PROGRAM MAIN
VAR
bChangeSeparatorToComma	: BOOL := TRUE;
P_TextModeWrite_WriteTrigger:BOOL:=FALSE;
P_TextModeWrite_WriteFilePath:T_MaxString := 'C:\Users\Administrator\Desktop\Pos.csv';
P_TextModeRead_ReadTrigger:BOOL:=FALSE;
P_TextModeRead_ReadFilePath:T_MaxString := 'C:\Users\Administrator\Desktop\Pos.csv';

CurrentJob: INT:= 0;//Job Code
CurrentJobState:STRING(80);//Say in which state

LAMP:BOOL;
POWER:BOOL;
Move_AB:BOOL;

SetPointGenEnable:ARRAY [0..5] OF MC_ExtSetPointGenEnable;
SetpointGenDisable:ARRAY [0..5] OF MC_ExtSetpointGenDisable;
SetPointGenEnable_output: ARRAY [0..5] OF ST_McOutputs;
SetPointGenDisable_output: ARRAY [0..5] OF ST_McOutputs;
enable:ARRAY [0..5] OF BOOL;
disable:ARRAY [0..5] OF BOOL;

position:ARRAY [0..5] OF LREAL;
velocity:ARRAY [0..5] OF LREAL;
direction:ARRAY [0..5] OF DINT;
acceleration:ARRAY [0..5] OF LREAL;

Pos_arr1:ARRAY[0..4999,0..5] OF LREAL;
i:INT;
FiFo_GetDimension: FiFoGetDimension;
fifo_display: STRING(255);

FiFo_GroupIntegrate1,FiFo_GroupIntegrate2,FiFo_GroupIntegrate3,FiFo_GroupIntegrate4,FiFo_GroupIntegrate6,FiFo_GroupIntegrate5: FiFoGroupIntegrate;
FiFo_SetChannelOverride:FiFoSetChannelOverride;
FiFo_Groupout1,FiFo_Groupout2,FiFo_Groupout3,FiFo_Groupout4,FiFo_Groupout5,FiFo_Groupout6,FiFo_Disintegrate,FiFo_Override_output:st_mcoutputs;
integrate_do:BOOL;
FiFo_GroupDisintegrate:FiFoGroupDisintegrate;

FiFo_Start:FiFoStart;
start_do:BOOL;
FiFo_Stop:FiFoStop;
stop_do:BOOL;
fifo_startoutput,fifo_stopoutput:st_mcoutputs;

FiFo_Write:FiFoWrite;
FIFO_write_do:BOOL;
FiFo_overWrite:FiFoOverwrite;
FIFO_overwrite_do:BOOL;
FIFO_write_output:st_mcoutputs;

END_VAR
VAR CONSTANT
	GlobalSetSpeed : ARRAY[0..5]OF LREAL:=[3200,3200,3200,3200,3200,3200];
END_VAR

IF bChangeSeparatorToComma THEN
	DEFAULT_CSV_FIELD_SEP := 16#2C;(* Comma ASCII code *)
ELSE
	DEFAULT_CSV_FIELD_SEP := 16#3B;(* Semicolon ASCII code *)
END_IF

IF FiFo_GetDimension.iNoOfAxes=6 AND FiFo_GetDimension.iNoOfFifoEntries=200 THEN
	fifo_display:='Parameters OK';
ELSE
	fifo_display:='Parameters Bad';
END_IF

//fifo();

GVL.LineMoveSpeed:=STRING_TO_LREAL(GVL.LineMoveSpeedString);
GVL.CMoveSpeed:=STRING_TO_LREAL(GVL.CMoveSpeedString);
GVL.OutMovePos[0]:=STRING_TO_LREAL(GVL.OutMovePosString[0]);
GVL.OutMovePos[1]:=STRING_TO_LREAL(GVL.OutMovePosString[1]);
GVL.OutMovePos[2]:=STRING_TO_LREAL(GVL.OutMovePosString[2]);
GVL.OutCMovePos[0]:=STRING_TO_LREAL(GVL.OutCMovePosString[0]);
GVL.OutCMovePos[1]:=STRING_TO_LREAL(GVL.OutCMovePosString[1]);
GVL.OutCMovePos[2]:=STRING_TO_LREAL(GVL.OutCMovePosString[2]);
GVL.MoveA[0]:=STRING_TO_LREAL(GVL.MoveAString[0])*24.995;
GVL.MoveA[1]:=STRING_TO_LREAL(GVL.MoveAString[1])*32.28;
GVL.MoveA[2]:=STRING_TO_LREAL(GVL.MoveAString[2])*49.845;
GVL.MoveA[3]:=STRING_TO_LREAL(GVL.MoveAString[3])*50.905;
GVL.MoveA[4]:=STRING_TO_LREAL(GVL.MoveAString[4])*80.34;
GVL.MoveA[5]:=STRING_TO_LREAL(GVL.MoveAString[5])*60.5;
GVL.OutActPos[0]:=-GVL.Axis[0].NcToPlc.ActPos/24.995;
GVL.OutActPos[1]:=-GVL.Axis[1].NcToPlc.ActPos/32.28;
GVL.OutActPos[2]:=GVL.Axis[2].NcToPlc.ActPos/49.845;
GVL.OutActPos[3]:=GVL.Axis[3].NcToPlc.ActPos/50.905;
GVL.OutActPos[4]:=GVL.Axis[4].NcToPlc.ActPos/80.34;
GVL.OutActPos[5]:=GVL.Axis[5].NcToPlc.ActPos/60.5;

IF GVL.ExtPosReady = FALSE THEN	
MC_ExtSetPointGenFeed(Position:=-GVL.OutActPos[0]*24.995,Velocity:= 0,Acceleration:=0,Direction:=1,Axis:=Axis[0]);	
MC_ExtSetPointGenFeed(Position:=-GVL.OutActPos[1]*32.28,Velocity:= 0,Acceleration:=0,Direction:=1,Axis:=Axis[1]);		
MC_ExtSetPointGenFeed(Position:=GVL.OutActPos[2]*49.845,Velocity:= 0,Acceleration:=0,Direction:=1,Axis:=Axis[2]);		
MC_ExtSetPointGenFeed(Position:=GVL.OutActPos[3]*50.905,Velocity:= 0,Acceleration:=0,Direction:=1,Axis:=Axis[3]);		
MC_ExtSetPointGenFeed(Position:=GVL.OutActPos[4]*80.34,Velocity:= 0,Acceleration:=0,Direction:=1,Axis:=Axis[4]);		
MC_ExtSetPointGenFeed(Position:=GVL.OutActPos[5]*60.5,Velocity:= 0,Acceleration:=0,Direction:=1,Axis:=Axis[5]);		
END_IF

CASE CurrentJob OF	
	0://None state
		AxisStopTrigger[0]:=FALSE;AxisStopTrigger[1]:=FALSE;AxisStopTrigger[2]:=FALSE;
		AxisStopTrigger[3]:=FALSE;AxisStopTrigger[4]:=FALSE;AxisStopTrigger[5]:=FALSE;
		AxisStop();//失能功能块
		
		JogFw[0]:=FALSE;JogFw[1]:=FALSE;JogFw[2]:=FALSE;JogFw[3]:=FALSE;JogFw[4]:=FALSE;JogFw[5]:=FALSE;
		JogBw[0]:=FALSE;JogBw[1]:=FALSE;JogBw[2]:=FALSE;JogBw[3]:=FALSE;JogBw[4]:=FALSE;JogBw[5]:=FALSE;
		Move_JOG();//失能功能块
		
		AxisMoveTrigger[0]:=FALSE;AxisMoveTrigger[1]:=FALSE;AxisMoveTrigger[2]:=FALSE;
		AxisMoveTrigger[3]:=FALSE;AxisMoveTrigger[4]:=FALSE;AxisMoveTrigger[5]:=FALSE;
		AxisMoveAbsoulte();//失能功能块
		
		Home[0]:=FALSE;Home[1]:=FALSE;Home[2]:=FALSE;
		Home[3]:=FALSE;Home[4]:=FALSE;Home[5]:=FALSE;
		Homing();//失能功能块	

		AxisResetTrigger[0]:=FALSE;AxisResetTrigger[1]:=FALSE;AxisResetTrigger[2]:=FALSE;
		AxisResetTrigger[3]:=FALSE;AxisResetTrigger[4]:=FALSE;AxisResetTrigger[5]:=FALSE;
		AxisReset();//失能功能块
		
		P_TextModeWrite_WriteTrigger:=FALSE;
		P_TextModeWrite();	
		P_TextModeRead_ReadTrigger:=FALSE;
		P_TextModeRead();//失能功能块
		
		SetPointGenEnable[0].Execute:=FALSE;SetPointGenEnable[1].Execute:=FALSE;
		SetPointGenEnable[2].Execute:=FALSE;SetPointGenEnable[3].Execute:=FALSE;
		SetPointGenEnable[4].Execute:=FALSE;SetPointGenEnable[5].Execute:=FALSE;

		SetPointGenDisable[0].Execute:=FALSE;SetPointGenDisable[1].Execute:=FALSE;		
		SetPointGenDisable[2].Execute:=FALSE;SetPointGenDisable[3].Execute:=FALSE;		
		SetPointGenDisable[4].Execute:=FALSE;SetPointGenDisable[5].Execute:=FALSE;		
		setpositionGen();
		
		JogMode[0]:=MC_JOGMODE_STANDARD_FAST;
		JogMode[1]:=MC_JOGMODE_STANDARD_FAST;
		JogMode[2]:=MC_JOGMODE_STANDARD_FAST;
		JogMode[3]:=MC_JOGMODE_STANDARD_FAST;
		JogMode[4]:=MC_JOGMODE_STANDARD_FAST;
		JogMode[5]:=MC_JOGMODE_STANDARD_FAST;

		GVL.KineModuleJob:=0;
	
		CurrentJobState:='Wait Command';
		i:=0;
	1://SetZero
		Home[0]:=TRUE;Home[1]:=TRUE;Home[2]:=TRUE;
		Home[3]:=TRUE;Home[4]:=TRUE;Home[5]:=TRUE;
		Home_Mode[0]:=MC_Direct;Home_Mode[1]:=MC_Direct;Home_Mode[2]:=MC_Direct;
		Home_Mode[3]:=MC_Direct;Home_Mode[4]:=MC_Direct;Home_Mode[5]:=MC_Direct;
		Home_Pos[0]:=0;Home_Pos[1]:=0;Home_Pos[2]:=0;
		Home_Pos[3]:=0;Home_Pos[4]:=0;Home_Pos[5]:=0;
		Homing();

		IF Home_Done[0]=TRUE AND 
		   Home_Done[1]=TRUE AND 
		   Home_Done[2]=TRUE AND 
		   Home_Done[3]=TRUE AND 
		   Home_Done[4]=TRUE AND 
		   Home_Done[5]=TRUE THEN
			CurrentJob:=0;
			CurrentJobState:='Set Origin Done!';
		ELSE
			CurrentJobState:='Set Origin Doing';
		END_IF
	2://直线插补
		setpointgenenable[0].Execute:=TRUE;setpointgenenable[1].Execute:=TRUE;
		setpointgenenable[2].Execute:=TRUE;setpointgenenable[3].Execute:=TRUE;
		setpointgenenable[4].Execute:=TRUE;setpointgenenable[5].Execute:=TRUE;
		IF  SetPointGenEnable[0].Enabled AND
			SetPointGenEnable[1].Enabled AND
			SetPointGenEnable[2].Enabled AND
			SetPointGenEnable[3].Enabled AND
			SetPointGenEnable[4].Enabled AND
			SetPointGenEnable[5].Enabled THEN
			
			i:=i+1;
			//IF(GVL.ExtPosOK = TRUE) THEN
			IF i > Pos_arr1[4999,5]+5 THEN
				SetPointGenDisable[0].Execute:=TRUE;SetPointGenDisable[1].Execute:=TRUE;
				SetPointGenDisable[2].Execute:=TRUE;SetPointGenDisable[3].Execute:=TRUE;
				SetPointGenDisable[4].Execute:=TRUE;SetPointGenDisable[5].Execute:=TRUE;
				setpositionGen();
				CurrentJob:=0;
			ELSE
				MC_ExtSetPointGenFeed(Position:=-Pos_arr1[i,5]*24.995,Velocity:= 0,Acceleration:=0,Direction:=1,Axis:=Axis[0]);
			
				MC_ExtSetPointGenFeed(Position:=-Pos_arr1[i,4]*32.28,Velocity:= 0,Acceleration:=0,Direction:=1,Axis:=Axis[1]);
			
				MC_ExtSetPointGenFeed(Position:=Pos_arr1[i,3]*49.845,Velocity:= 0,Acceleration:=0,Direction:=1,Axis:=Axis[2]);
			
				MC_ExtSetPointGenFeed(Position:=Pos_arr1[i,2]*50.905,Velocity:= 0,Acceleration:=0,Direction:=1,Axis:=Axis[3]);
			
				MC_ExtSetPointGenFeed(Position:=Pos_arr1[i,1]*80.34,Velocity:= 0,Acceleration:=0,Direction:=1,Axis:=Axis[4]);
			
				MC_ExtSetPointGenFeed(Position:=Pos_arr1[i,0]*60.5,Velocity:= 0,Acceleration:=0,Direction:=1,Axis:=Axis[5]);
			END_IF
			//GVL.KineModuleJob:=4;
			//IF GVL.ExtPosReady THEN
			//MC_ExtSetPointGenFeed(Position:=-ExtPos[0]*24.995,Velocity:= 0,Acceleration:=0,Direction:=1,Axis:=Axis[0]);
			
			//MC_ExtSetPointGenFeed(Position:=-ExtPos[1]*32.28,Velocity:= 0,Acceleration:=0,Direction:=1,Axis:=Axis[1]);
			
			//MC_ExtSetPointGenFeed(Position:=ExtPos[2]*49.845,Velocity:= 0,Acceleration:=0,Direction:=1,Axis:=Axis[2]);
			
			//MC_ExtSetPointGenFeed(Position:=ExtPos[3]*50.905,Velocity:= 0,Acceleration:=0,Direction:=1,Axis:=Axis[3]);
			
			//MC_ExtSetPointGenFeed(Position:=ExtPos[4]*80.34,Velocity:= 0,Acceleration:=0,Direction:=1,Axis:=Axis[4]);
			
			//MC_ExtSetPointGenFeed(Position:=ExtPos[5]*60.5,Velocity:= 0,Acceleration:=0,Direction:=1,Axis:=Axis[5]);		
			//END_IF
		END_IF
		setpositionGen();
	3://JogForward
		JogFw[axisNum]:=TRUE;
		Move_JOG();
		CurrentJob:=3;
		CurrentJobState:='Jog Forward';
	4://JogBackward
		JogBw[axisNum]:=TRUE;
		Move_JOG();
		CurrentJob:=4;
		CurrentJobState:='Jog Backward';
	5://Stop
		AxisStopDeceleration[0]:=15000;AxisStopDeceleration[1]:=15000;AxisStopDeceleration[2]:=15000;
		AxisStopDeceleration[3]:=15000;AxisStopDeceleration[4]:=15000;AxisStopDeceleration[5]:=15000;
		AxisStopTrigger[0]:=TRUE;AxisStopTrigger[1]:=TRUE;AxisStopTrigger[2]:=TRUE;
		AxisStopTrigger[3]:=TRUE;AxisStopTrigger[4]:=TRUE;AxisStopTrigger[5]:=TRUE;
		AxisStop();
		IF AxisStopDone[0]=TRUE AND
		   AxisStopDone[1]=TRUE AND
		   AxisStopDone[2]=TRUE AND
		   AxisStopDone[3]=TRUE AND
		   AxisStopDone[4]=TRUE AND
		   AxisStopDone[5]=TRUE THEN
			CurrentJobState:='Stop Done';
			CurrentJob:=0;
		ELSE
			CurrentJobState:='Stop Doing';
		END_IF
	6://Move To HOME
		AxisMovePosition[0]:=-3683.8943;AxisMovePosition[1]:=5173.9531;AxisMovePosition[2]:=318.8809;
		AxisMovePosition[3]:=5194.3991;AxisMovePosition[4]:=307.0219;AxisMovePosition[5]:=774.2587;	
		AxisMoveSpeed[0]:=2000;AxisMoveSpeed[1]:=2000;AxisMoveSpeed[2]:=2000;
		AxisMoveSpeed[3]:=2000;AxisMoveSpeed[4]:=2000;AxisMoveSpeed[5]:=2000;
		
		AxisMoveTrigger[0]:=TRUE;AxisMoveTrigger[1]:=TRUE;AxisMoveTrigger[2]:=TRUE;
		AxisMoveTrigger[3]:=TRUE;AxisMoveTrigger[4]:=TRUE;AxisMoveTrigger[5]:=TRUE;
		AxisMoveAbsoulte();
		
		IF AxisMoveAbsoluteDone[0]=TRUE AND 
		   AxisMoveAbsoluteDone[1]=TRUE AND 
		   AxisMoveAbsoluteDone[2]=TRUE AND 
		   AxisMoveAbsoluteDone[3]=TRUE AND 
		   AxisMoveAbsoluteDone[4]=TRUE AND 
		   AxisMoveAbsoluteDone[5]=TRUE THEN			
			CurrentJobState:='Home Done';
			CurrentJob:=1;			
		ELSE
			CurrentJobState:='Home Doing';
		END_IF
	7://Move To A
		AxisMovePosition[0]:=MoveA[0];AxisMovePosition[1]:=MoveA[1];AxisMovePosition[2]:=MoveA[2];
		AxisMovePosition[3]:=MoveA[3];AxisMovePosition[4]:=MoveA[4];AxisMovePosition[5]:=MoveA[5];
		
		AxisMoveSpeed[0]:=GlobalSetSpeed[0];AxisMoveSpeed[1]:=GlobalSetSpeed[1];AxisMoveSpeed[2]:=GlobalSetSpeed[2];
		AxisMoveSpeed[3]:=GlobalSetSpeed[3];AxisMoveSpeed[4]:=GlobalSetSpeed[4];AxisMoveSpeed[5]:=GlobalSetSpeed[5];
		
		AxisMoveTrigger[0]:=TRUE;AxisMoveTrigger[1]:=TRUE;AxisMoveTrigger[2]:=TRUE;
		AxisMoveTrigger[3]:=TRUE;AxisMoveTrigger[4]:=TRUE;AxisMoveTrigger[5]:=TRUE;
		AxisMoveAbsoulte();
		
		IF AxisMoveAbsoluteDone[0]=TRUE AND 
		   AxisMoveAbsoluteDone[1]=TRUE AND 
		   AxisMoveAbsoluteDone[2]=TRUE AND 
		   AxisMoveAbsoluteDone[3]=TRUE AND 
		   AxisMoveAbsoluteDone[4]=TRUE AND 
		   AxisMoveAbsoluteDone[5]=TRUE THEN		
			CurrentJobState:='MOVE A Done';
			CurrentJob:=0;		
		ELSE
			CurrentJobState:='MOVE A Doing';
		END_IF
	8://往复运动
		IF Move_AB=FALSE THEN
		//AxisMovePosition[0]:=-742579.6646;AxisMovePosition[1]:=5125.997925;AxisMovePosition[2]:=223.8519;
		//AxisMovePosition[3]:=5161.5829;AxisMovePosition[4]:=-31.9675;AxisMovePosition[5]:=774.2587;	
		AxisMovePosition[0]:=0;AxisMovePosition[1]:=0;AxisMovePosition[2]:=0;
		AxisMovePosition[3]:=0;AxisMovePosition[4]:=0;AxisMovePosition[5]:=0;
		ELSE
		AxisMovePosition[0]:=MoveA[0];AxisMovePosition[1]:=MoveA[1];AxisMovePosition[2]:=MoveA[2];
		AxisMovePosition[3]:=MoveA[3];AxisMovePosition[4]:=MoveA[4];AxisMovePosition[5]:=MoveA[5];	
		END_IF
		AxisMoveSpeed[0]:=2000;AxisMoveSpeed[1]:=2000;AxisMoveSpeed[2]:=2000;
		AxisMoveSpeed[3]:=2000;AxisMoveSpeed[4]:=2000;AxisMoveSpeed[5]:=2000;
		
		AxisMoveTrigger[0]:=TRUE;AxisMoveTrigger[1]:=TRUE;AxisMoveTrigger[2]:=TRUE;
		AxisMoveTrigger[3]:=TRUE;AxisMoveTrigger[4]:=TRUE;AxisMoveTrigger[5]:=TRUE;
		AxisMoveAbsoulte();
		
		IF AxisMoveAbsoluteDone[0]=TRUE AND 
		   AxisMoveAbsoluteDone[1]=TRUE AND 
		   AxisMoveAbsoluteDone[2]=TRUE AND 
		   AxisMoveAbsoluteDone[3]=TRUE AND 
		   AxisMoveAbsoluteDone[4]=TRUE AND 
		   AxisMoveAbsoluteDone[5]=TRUE THEN	
		   Move_AB:= NOT Move_AB;
		   AxisMoveTrigger[0]:=FALSE;AxisMoveTrigger[1]:=FALSE;AxisMoveTrigger[2]:=FALSE;
		   AxisMoveTrigger[3]:=FALSE;AxisMoveTrigger[4]:=FALSE;AxisMoveTrigger[5]:=FALSE;
		   AxisMoveAbsoulte();//失能功能块
		END_IF
		CurrentJobState:='Reciprocating Doing';
	9://复位
		AxisResetTrigger[0]:=TRUE;AxisResetTrigger[1]:=TRUE;AxisResetTrigger[2]:=TRUE;
		AxisResetTrigger[3]:=TRUE;AxisResetTrigger[4]:=TRUE;AxisResetTrigger[5]:=TRUE;
		AxisReset();
		IF AxisResetDone[0]=TRUE AND
		   AxisResetDone[1]=TRUE AND
		   AxisResetDone[2]=TRUE AND
		   AxisResetDone[3]=TRUE AND
		   AxisResetDone[4]=TRUE AND
		   AxisResetDone[5]=TRUE THEN	
			CurrentJobState:='Axis Reset Done';
			CurrentJob:=0;
		ELSE
			CurrentJobState:='Axis Reset Doing';
		END_IF
	10://read csv
		//P_TextModeRead_ReadTrigger:=TRUE;
		//CurrentJobState:='Read CSV';
		//P_TextModeRead();
		GVL.KineModuleJob:=2;
		CurrentJob:=0;
	11://Move to origin
		AxisMovePosition[0]:=0;AxisMovePosition[1]:=0;AxisMovePosition[2]:=0;
		AxisMovePosition[3]:=0;AxisMovePosition[4]:=0;AxisMovePosition[5]:=0;
		
		AxisMoveSpeed[0]:=2000;AxisMoveSpeed[1]:=2000;AxisMoveSpeed[2]:=2000;
		AxisMoveSpeed[3]:=2000;AxisMoveSpeed[4]:=2000;AxisMoveSpeed[5]:=2000;
		
		AxisMoveTrigger[0]:=TRUE;AxisMoveTrigger[1]:=TRUE;AxisMoveTrigger[2]:=TRUE;
		AxisMoveTrigger[3]:=TRUE;AxisMoveTrigger[4]:=TRUE;AxisMoveTrigger[5]:=TRUE;
		AxisMoveAbsoulte();
		
		IF AxisMoveAbsoluteDone[0]=TRUE AND 
		   AxisMoveAbsoluteDone[1]=TRUE AND 
		   AxisMoveAbsoluteDone[2]=TRUE AND 
		   AxisMoveAbsoluteDone[3]=TRUE AND 
		   AxisMoveAbsoluteDone[4]=TRUE AND 
		   AxisMoveAbsoluteDone[5]=TRUE THEN		
			CurrentJobState:='MOVE Origin Done';
			CurrentJob:=0;		
		ELSE
			CurrentJobState:='MOVE Origin Doing';
		END_IF
	12://直线插补
		setpointgenenable[0].Execute:=TRUE;setpointgenenable[1].Execute:=TRUE;
		setpointgenenable[2].Execute:=TRUE;setpointgenenable[3].Execute:=TRUE;
		setpointgenenable[4].Execute:=TRUE;setpointgenenable[5].Execute:=TRUE;
		IF  SetPointGenEnable[0].Enabled AND
			SetPointGenEnable[1].Enabled AND
			SetPointGenEnable[2].Enabled AND
			SetPointGenEnable[3].Enabled AND
			SetPointGenEnable[4].Enabled AND
			SetPointGenEnable[5].Enabled THEN
			
			IF(GVL.ExtPosOK = TRUE) THEN			
				SetPointGenDisable[0].Execute:=TRUE;SetPointGenDisable[1].Execute:=TRUE;
				SetPointGenDisable[2].Execute:=TRUE;SetPointGenDisable[3].Execute:=TRUE;
				SetPointGenDisable[4].Execute:=TRUE;SetPointGenDisable[5].Execute:=TRUE;
				setpositionGen();
				CurrentJob:=0;
			END_IF
			
			GVL.KineModuleJob:=3;
			IF GVL.ExtPosReady THEN
			MC_ExtSetPointGenFeed(Position:=ExtPos[0]*24.995,Velocity:= 0,Acceleration:=0,Direction:=1,Axis:=Axis[0]);
			
			MC_ExtSetPointGenFeed(Position:=-ExtPos[1]*32.28,Velocity:= 0,Acceleration:=0,Direction:=1,Axis:=Axis[1]);
			
			MC_ExtSetPointGenFeed(Position:=ExtPos[2]*49.845,Velocity:= 0,Acceleration:=0,Direction:=1,Axis:=Axis[2]);
			
			MC_ExtSetPointGenFeed(Position:=ExtPos[3]*50.905,Velocity:= 0,Acceleration:=0,Direction:=1,Axis:=Axis[3]);
			
			MC_ExtSetPointGenFeed(Position:=ExtPos[4]*80.34,Velocity:= 0,Acceleration:=0,Direction:=1,Axis:=Axis[4]);
			
			MC_ExtSetPointGenFeed(Position:=ExtPos[5]*60.5,Velocity:= 0,Acceleration:=0,Direction:=1,Axis:=Axis[5]);		
			END_IF
		END_IF
		setpositionGen();
	13://关节空间运动
		GVL.KineModuleJob:=1;
		CurrentJob:=0;
END_CASE

//错误检测
IF  AxisPowerError[0] OR
	AxisPowerError[1] OR
	AxisPowerError[2] OR
	AxisPowerError[3] OR
	AxisPowerError[4] OR
	AxisPowerError[5] THEN
	//POWER:=FALSE;
	CurrentJob:=9;
END_IF
//电机上下电
IF POWER=TRUE THEN
	AxisPowerTrigger[0]:=TRUE;
	AxisPowerTrigger[1]:=TRUE;
	AxisPowerTrigger[2]:=TRUE;
	AxisPowerTrigger[3]:=TRUE;
	AxisPowerTrigger[4]:=TRUE;
	AxisPowerTrigger[5]:=TRUE;
	AxisEnable();
	IF  AxisPowerReady[0]=TRUE AND 
		AxisPowerReady[1]=TRUE AND 
		AxisPowerReady[2]=TRUE AND 
		AxisPowerReady[3]=TRUE AND
		AxisPowerReady[4]=TRUE AND 
		AxisPowerReady[5]=TRUE THEN
		LAMP:=TRUE;
	END_IF
ELSE
	AxisPowerTrigger[0]:=FALSE;
	AxisPowerTrigger[1]:=FALSE;
	AxisPowerTrigger[2]:=FALSE;
	AxisPowerTrigger[3]:=FALSE;
	AxisPowerTrigger[4]:=FALSE;
	AxisPowerTrigger[5]:=FALSE;
	AxisEnable();
	IF  AxisPowerReady[0]=FALSE AND
		AxisPowerReady[1]=FALSE AND
		AxisPowerReady[2]=FALSE AND
		AxisPowerReady[3]=FALSE AND
		AxisPowerReady[4]=FALSE AND
		AxisPowerReady[5]=FALSE THEN
		LAMP:=FALSE;   
	END_IF
END_IF

ACTION fifo:
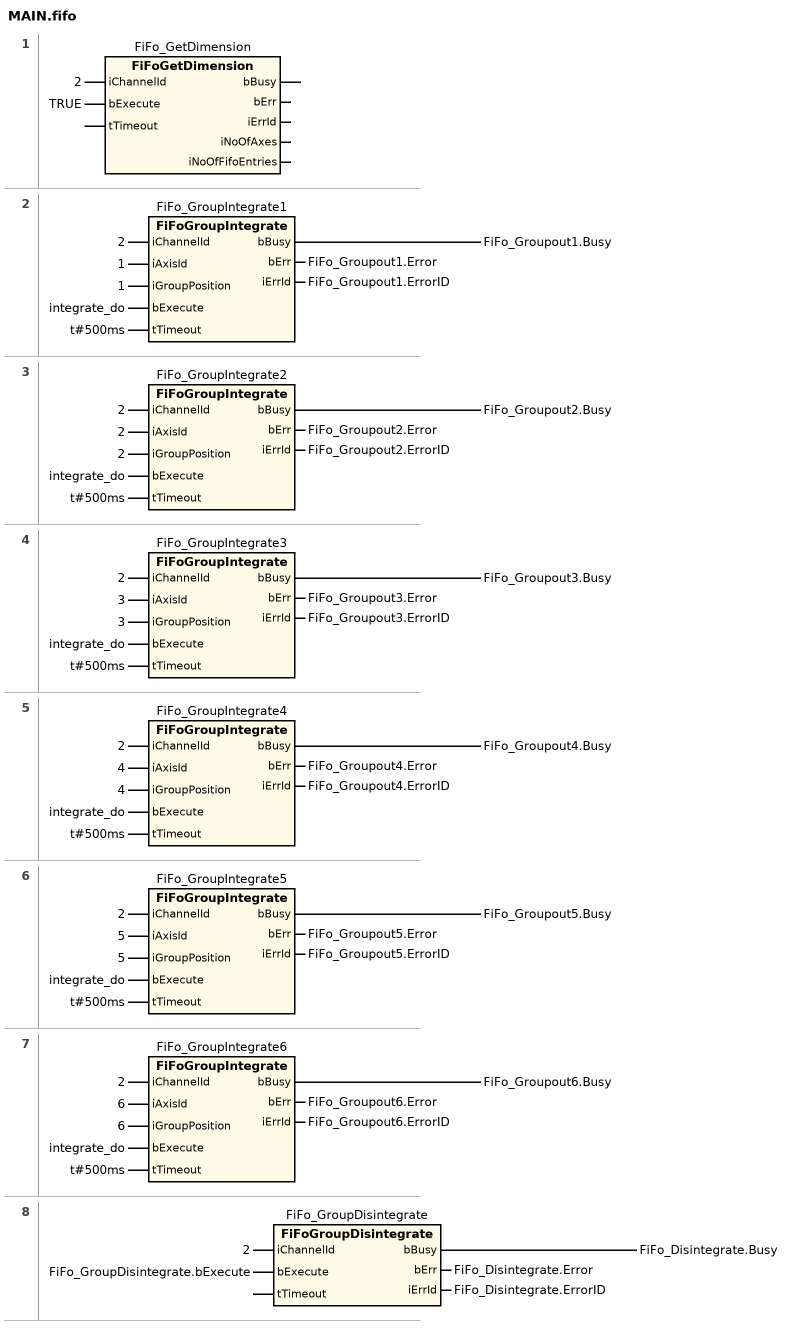
// NETWORK 1
FiFo_GetDimension(iChannelId := 2, bExecute := TRUE); // FiFoGetDimension

// NETWORK 2
FiFo_GroupIntegrate1(
    iChannelId := 2,
    iAxisId := 1,
    iGroupPosition := 1,
    bExecute := integrate_do,
    tTimeout := t#500ms,
    bErr => FiFo_Groupout1.Error,
    iErrId => FiFo_Groupout1.ErrorID); // FiFoGroupIntegrate
FiFo_Groupout1.Busy := FiFo_GroupIntegrate1.bBusy;

// NETWORK 3
FiFo_GroupIntegrate2(
    iChannelId := 2,
    iAxisId := 2,
    iGroupPosition := 2,
    bExecute := integrate_do,
    tTimeout := t#500ms,
    bErr => FiFo_Groupout2.Error,
    iErrId => FiFo_Groupout2.ErrorID); // FiFoGroupIntegrate
FiFo_Groupout2.Busy := FiFo_GroupIntegrate2.bBusy;

// NETWORK 4
FiFo_GroupIntegrate3(
    iChannelId := 2,
    iAxisId := 3,
    iGroupPosition := 3,
    bExecute := integrate_do,
    tTimeout := t#500ms,
    bErr => FiFo_Groupout3.Error,
    iErrId => FiFo_Groupout3.ErrorID); // FiFoGroupIntegrate
FiFo_Groupout3.Busy := FiFo_GroupIntegrate3.bBusy;

// NETWORK 5
FiFo_GroupIntegrate4(
    iChannelId := 2,
    iAxisId := 4,
    iGroupPosition := 4,
    bExecute := integrate_do,
    tTimeout := t#500ms,
    bErr => FiFo_Groupout4.Error,
    iErrId => FiFo_Groupout4.ErrorID); // FiFoGroupIntegrate
FiFo_Groupout4.Busy := FiFo_GroupIntegrate4.bBusy;

// NETWORK 6
FiFo_GroupIntegrate5(
    iChannelId := 2,
    iAxisId := 5,
    iGroupPosition := 5,
    bExecute := integrate_do,
    tTimeout := t#500ms,
    bErr => FiFo_Groupout5.Error,
    iErrId => FiFo_Groupout5.ErrorID); // FiFoGroupIntegrate
FiFo_Groupout5.Busy := FiFo_GroupIntegrate5.bBusy;

// NETWORK 7
FiFo_GroupIntegrate6(
    iChannelId := 2,
    iAxisId := 6,
    iGroupPosition := 6,
    bExecute := integrate_do,
    tTimeout := t#500ms,
    bErr => FiFo_Groupout6.Error,
    iErrId => FiFo_Groupout6.ErrorID); // FiFoGroupIntegrate
FiFo_Groupout6.Busy := FiFo_GroupIntegrate6.bBusy;

// NETWORK 8
FiFo_GroupDisintegrate(
    iChannelId := 2,
    bExecute := FiFo_GroupDisintegrate.bExecute,
    bErr => FiFo_Disintegrate.Error,
    iErrId => FiFo_Disintegrate.ErrorID); // FiFoGroupDisintegrate
FiFo_Disintegrate.Busy := FiFo_GroupDisintegrate.bBusy;

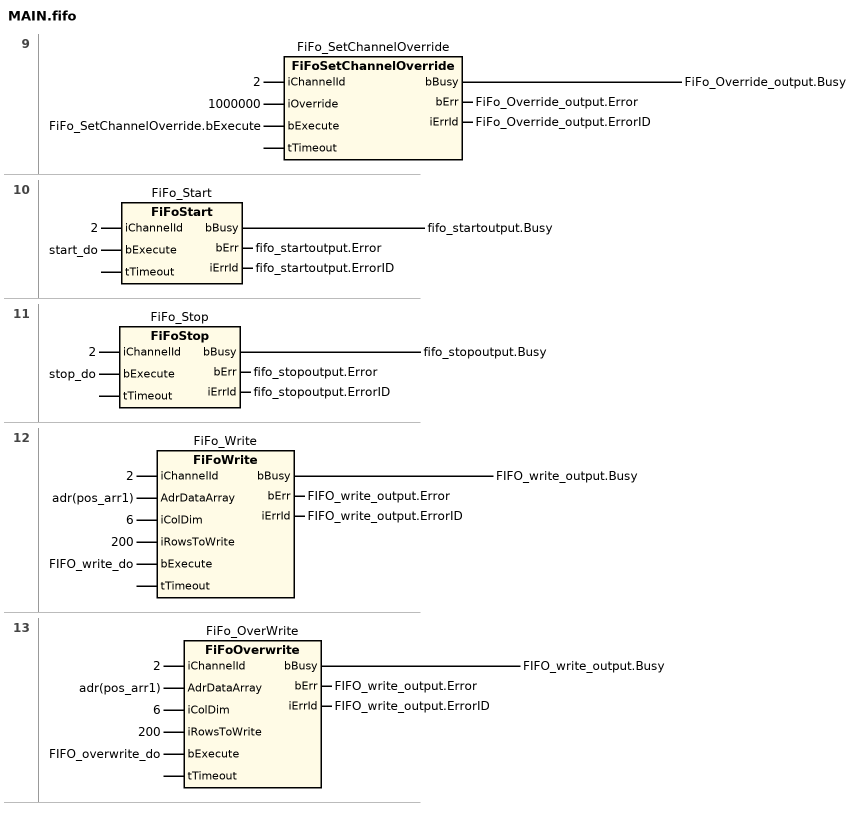
// NETWORK 9
FiFo_SetChannelOverride(
    iChannelId := 2,
    iOverride := 1000000,
    bExecute := FiFo_SetChannelOverride.bExecute,
    bErr => FiFo_Override_output.Error,
    iErrId => FiFo_Override_output.ErrorID); // FiFoSetChannelOverride
FiFo_Override_output.Busy := FiFo_SetChannelOverride.bBusy;

// NETWORK 10
FiFo_Start(
    iChannelId := 2,
    bExecute := start_do,
    bErr => fifo_startoutput.Error,
    iErrId => fifo_startoutput.ErrorID); // FiFoStart
fifo_startoutput.Busy := FiFo_Start.bBusy;

// NETWORK 11
FiFo_Stop(
    iChannelId := 2,
    bExecute := stop_do,
    bErr => fifo_stopoutput.Error,
    iErrId => fifo_stopoutput.ErrorID); // FiFoStop
fifo_stopoutput.Busy := FiFo_Stop.bBusy;

// NETWORK 12
FiFo_Write(
    iChannelId := 2,
    AdrDataArray := adr(pos_arr1),
    iColDim := 6,
    iRowsToWrite := 200,
    bExecute := FIFO_write_do,
    bErr => FIFO_write_output.Error,
    iErrId => FIFO_write_output.ErrorID); // FiFoWrite
FIFO_write_output.Busy := FiFo_Write.bBusy;

// NETWORK 13
FiFo_OverWrite(
    iChannelId := 2,
    AdrDataArray := adr(pos_arr1),
    iColDim := 6,
    iRowsToWrite := 200,
    bExecute := FIFO_overwrite_do,
    bErr => FIFO_write_output.Error,
    iErrId => FIFO_write_output.ErrorID); // FiFoOverwrite
FIFO_write_output.Busy := FiFo_OverWrite.bBusy;
END_ACTION

ACTION setpositionGen:
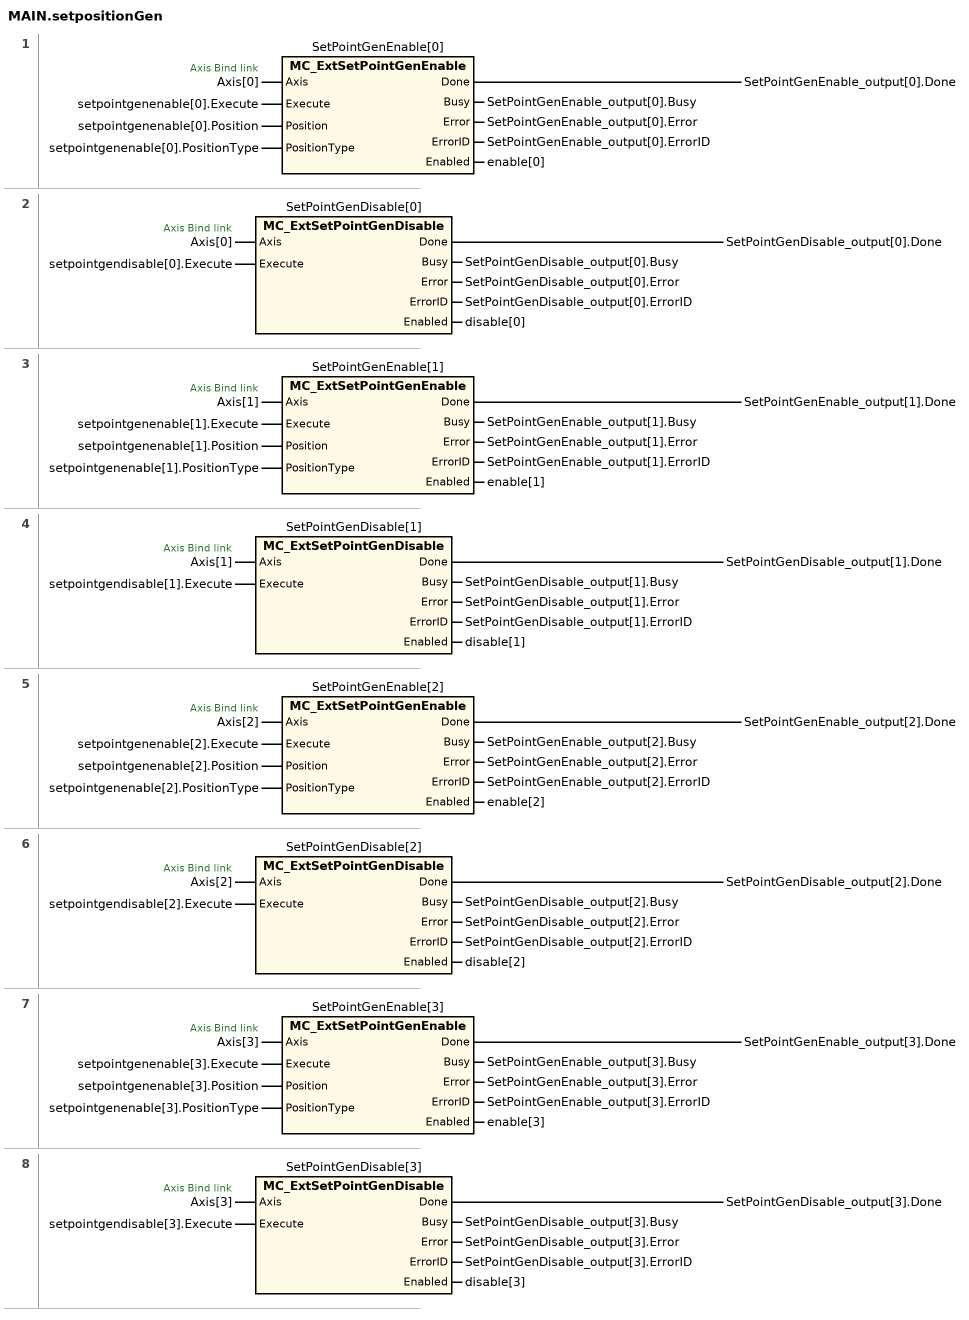
// NETWORK 1
//   Axis[0]: Axis Bind link
SetPointGenEnable[0](
    Axis := Axis[0],
    Execute := setpointgenenable[0].Execute,
    Position := setpointgenenable[0].Position,
    PositionType := setpointgenenable[0].PositionType,
    Busy => SetPointGenEnable_output[0].Busy,
    Error => SetPointGenEnable_output[0].Error,
    ErrorID => SetPointGenEnable_output[0].ErrorID,
    Enabled => enable[0]); // MC_ExtSetPointGenEnable
SetPointGenEnable_output[0].Done := SetPointGenEnable[0].Done;

// NETWORK 2
//   Axis[0]: Axis Bind link
SetPointGenDisable[0](
    Axis := Axis[0],
    Execute := setpointgendisable[0].Execute,
    Busy => SetPointGenDisable_output[0].Busy,
    Error => SetPointGenDisable_output[0].Error,
    ErrorID => SetPointGenDisable_output[0].ErrorID,
    Enabled => disable[0]); // MC_ExtSetPointGenDisable
SetPointGenDisable_output[0].Done := SetPointGenDisable[0].Done;

// NETWORK 3
//   Axis[1]: Axis Bind link
SetPointGenEnable[1](
    Axis := Axis[1],
    Execute := setpointgenenable[1].Execute,
    Position := setpointgenenable[1].Position,
    PositionType := setpointgenenable[1].PositionType,
    Busy => SetPointGenEnable_output[1].Busy,
    Error => SetPointGenEnable_output[1].Error,
    ErrorID => SetPointGenEnable_output[1].ErrorID,
    Enabled => enable[1]); // MC_ExtSetPointGenEnable
SetPointGenEnable_output[1].Done := SetPointGenEnable[1].Done;

// NETWORK 4
//   Axis[1]: Axis Bind link
SetPointGenDisable[1](
    Axis := Axis[1],
    Execute := setpointgendisable[1].Execute,
    Busy => SetPointGenDisable_output[1].Busy,
    Error => SetPointGenDisable_output[1].Error,
    ErrorID => SetPointGenDisable_output[1].ErrorID,
    Enabled => disable[1]); // MC_ExtSetPointGenDisable
SetPointGenDisable_output[1].Done := SetPointGenDisable[1].Done;

// NETWORK 5
//   Axis[2]: Axis Bind link
SetPointGenEnable[2](
    Axis := Axis[2],
    Execute := setpointgenenable[2].Execute,
    Position := setpointgenenable[2].Position,
    PositionType := setpointgenenable[2].PositionType,
    Busy => SetPointGenEnable_output[2].Busy,
    Error => SetPointGenEnable_output[2].Error,
    ErrorID => SetPointGenEnable_output[2].ErrorID,
    Enabled => enable[2]); // MC_ExtSetPointGenEnable
SetPointGenEnable_output[2].Done := SetPointGenEnable[2].Done;

// NETWORK 6
//   Axis[2]: Axis Bind link
SetPointGenDisable[2](
    Axis := Axis[2],
    Execute := setpointgendisable[2].Execute,
    Busy => SetPointGenDisable_output[2].Busy,
    Error => SetPointGenDisable_output[2].Error,
    ErrorID => SetPointGenDisable_output[2].ErrorID,
    Enabled => disable[2]); // MC_ExtSetPointGenDisable
SetPointGenDisable_output[2].Done := SetPointGenDisable[2].Done;

// NETWORK 7
//   Axis[3]: Axis Bind link
SetPointGenEnable[3](
    Axis := Axis[3],
    Execute := setpointgenenable[3].Execute,
    Position := setpointgenenable[3].Position,
    PositionType := setpointgenenable[3].PositionType,
    Busy => SetPointGenEnable_output[3].Busy,
    Error => SetPointGenEnable_output[3].Error,
    ErrorID => SetPointGenEnable_output[3].ErrorID,
    Enabled => enable[3]); // MC_ExtSetPointGenEnable
SetPointGenEnable_output[3].Done := SetPointGenEnable[3].Done;

// NETWORK 8
//   Axis[3]: Axis Bind link
SetPointGenDisable[3](
    Axis := Axis[3],
    Execute := setpointgendisable[3].Execute,
    Busy => SetPointGenDisable_output[3].Busy,
    Error => SetPointGenDisable_output[3].Error,
    ErrorID => SetPointGenDisable_output[3].ErrorID,
    Enabled => disable[3]); // MC_ExtSetPointGenDisable
SetPointGenDisable_output[3].Done := SetPointGenDisable[3].Done;

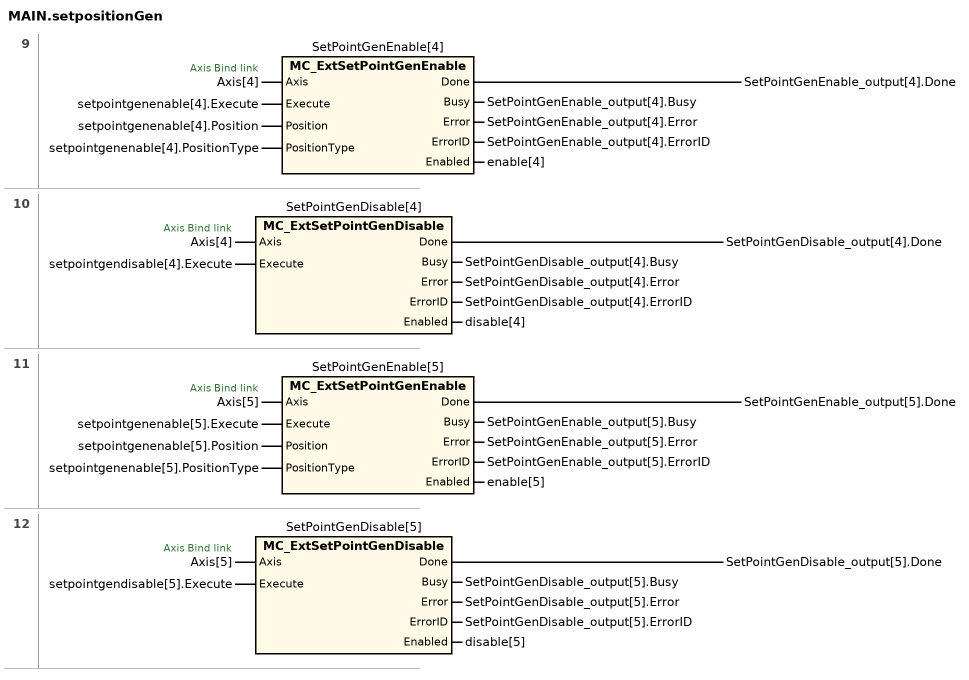
// NETWORK 9
//   Axis[4]: Axis Bind link
SetPointGenEnable[4](
    Axis := Axis[4],
    Execute := setpointgenenable[4].Execute,
    Position := setpointgenenable[4].Position,
    PositionType := setpointgenenable[4].PositionType,
    Busy => SetPointGenEnable_output[4].Busy,
    Error => SetPointGenEnable_output[4].Error,
    ErrorID => SetPointGenEnable_output[4].ErrorID,
    Enabled => enable[4]); // MC_ExtSetPointGenEnable
SetPointGenEnable_output[4].Done := SetPointGenEnable[4].Done;

// NETWORK 10
//   Axis[4]: Axis Bind link
SetPointGenDisable[4](
    Axis := Axis[4],
    Execute := setpointgendisable[4].Execute,
    Busy => SetPointGenDisable_output[4].Busy,
    Error => SetPointGenDisable_output[4].Error,
    ErrorID => SetPointGenDisable_output[4].ErrorID,
    Enabled => disable[4]); // MC_ExtSetPointGenDisable
SetPointGenDisable_output[4].Done := SetPointGenDisable[4].Done;

// NETWORK 11
//   Axis[5]: Axis Bind link
SetPointGenEnable[5](
    Axis := Axis[5],
    Execute := setpointgenenable[5].Execute,
    Position := setpointgenenable[5].Position,
    PositionType := setpointgenenable[5].PositionType,
    Busy => SetPointGenEnable_output[5].Busy,
    Error => SetPointGenEnable_output[5].Error,
    ErrorID => SetPointGenEnable_output[5].ErrorID,
    Enabled => enable[5]); // MC_ExtSetPointGenEnable
SetPointGenEnable_output[5].Done := SetPointGenEnable[5].Done;

// NETWORK 12
//   Axis[5]: Axis Bind link
SetPointGenDisable[5](
    Axis := Axis[5],
    Execute := setpointgendisable[5].Execute,
    Busy => SetPointGenDisable_output[5].Busy,
    Error => SetPointGenDisable_output[5].Error,
    ErrorID => SetPointGenDisable_output[5].ErrorID,
    Enabled => disable[5]); // MC_ExtSetPointGenDisable
SetPointGenDisable_output[5].Done := SetPointGenDisable[5].Done;
END_ACTION

END_PROGRAM

(* stored: Version 1.1.0.1, ProductVersion 3.1.4018.5
   POU MAIN: Id {5df62128-f8ca-4cb2-82f0-fb5ed1ffd77a}, SpecialFunc None
   Action fifo: Id {b02c1073-82f4-4223-8646-23a3528a33ec}
   Action setpositionGen: Id {ae6c9d44-33f1-4fe3-8a12-7ba33d831292} *)
